// Mitsubishi GX Works2 project: IHW4   PLC: Q03UDE

// global labels: Global1
VAR_GLOBAL
  START_BUTTON AT X50 : BOOL;
  STOP_BUTTON AT X51 : BOOL;
  SENSOR_A AT X53 : BOOL;
  SENSOR_B AT X54 : BOOL;
  SENSOR_C AT X55 : BOOL;
  SENSOR_D AT X56 : BOOL;
  CRANE_UP AT Y40 : BOOL;
  CRANE_DOWN AT Y41 : BOOL;
  CRANE_LEFT AT Y42 : BOOL;
  CRANE_RIGHT AT Y43 : BOOL;
  ESTOP_BUTTON AT X52 : BOOL;
END_VAR

PROGRAM MAIN
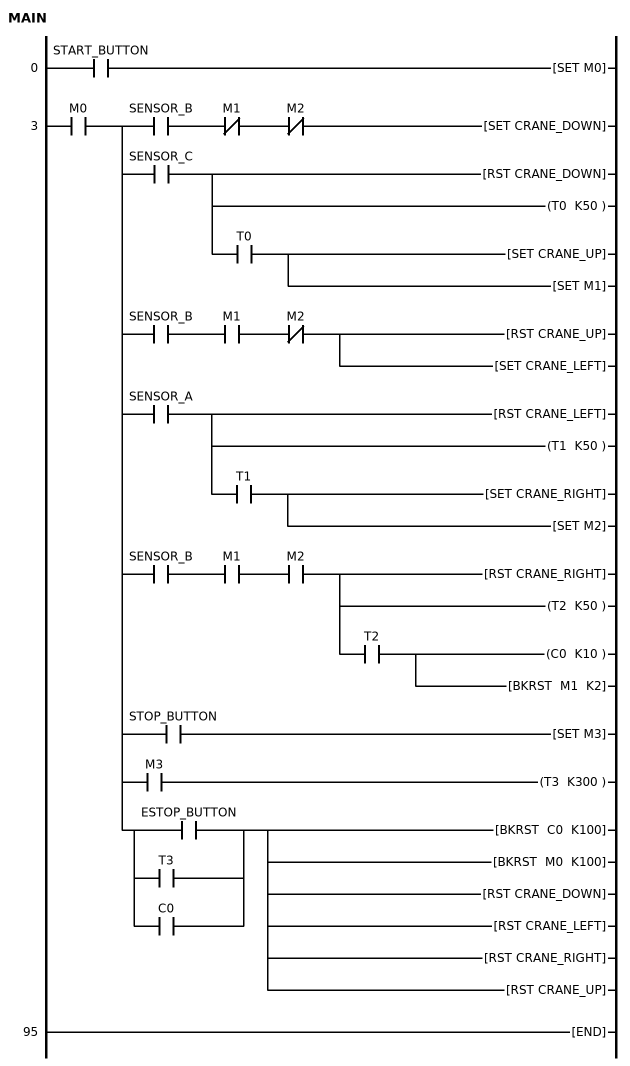
0     LD      START_BUTTON
      SET     M0
3     LD      M0
      MPS
      AND     SENSOR_B
      ANI     M1
      ANI     M2
      SET     CRANE_DOWN
      MRD
      AND     SENSOR_C
      RST     CRANE_DOWN
      OUT     T0 K50
      AND     T0
      SET     CRANE_UP
      SET     M1
      MRD
      AND     SENSOR_B
      AND     M1
      ANI     M2
      RST     CRANE_UP
      SET     CRANE_LEFT
      MRD
      AND     SENSOR_A
      RST     CRANE_LEFT
      OUT     T1 K50
      AND     T1
      SET     CRANE_RIGHT
      SET     M2
      MRD
      AND     SENSOR_B
      AND     M1
      AND     M2
      RST     CRANE_RIGHT
      OUT     T2 K50
      AND     T2
      OUT     C0 K10
      BKRST   M1 K2
      MRD
      AND     STOP_BUTTON
      SET     M3
      MRD
      AND     M3
      OUT     T3 K300
      MPP
      LD      ESTOP_BUTTON
      OR      T3
      OR      C0
      ANB
      BKRST   C0 K100
      BKRST   M0 K100
      RST     CRANE_DOWN
      RST     CRANE_LEFT
      RST     CRANE_RIGHT
      RST     CRANE_UP
95    END
END_PROGRAM
